{attribute 'enable_dynamic_creation'}
FUNCTION_BLOCK FB_JobEventStream IMPLEMENTS InterfaceJobEventObservable
VAR_INPUT
END_VAR
VAR_OUTPUT
END_VAR
VAR
	_observers : ARRAY[1..ParamFuturesLib.MAX_JOB_EVENT_OBSERVERS] OF InterfaceJobEventObserver;
	_filter_state : E_FutureExecutionState := E_FutureExecutionState.idle;
	_filter_event_type : E_JobEventType := E_JobEventType.TRANSITION;
	_filter_executor_id : T_MaxString := '';
	_filter_error_min : UDINT := 0;
	_filter_error_max : UDINT := 16#FFFFFFFF;
	_filter_enabled : ST_FilterStates;
END_VAR

METHOD ClearFilters : InterfaceJobEventObservable
VAR_INPUT
END_VAR
_filter_enabled.state := FALSE;
_filter_enabled.event_type := FALSE;
_filter_enabled.executor_id := FALSE;
_filter_enabled.error_range := FALSE;
ClearFilters := THIS^;
END_METHOD

METHOD emit_event : BOOL
VAR_INPUT
	event : ST_JobEvent;
END_VAR
VAR
	i : UINT;
	should_emit : BOOL := TRUE;
END_VAR
// フィルター判定
IF _filter_enabled.state AND event.state_new <> _filter_state THEN
	should_emit := FALSE;
END_IF
IF _filter_enabled.event_type AND event.event_type <> _filter_event_type THEN
	should_emit := FALSE;
END_IF
IF _filter_enabled.executor_id AND event.executor_id <> _filter_executor_id THEN
	should_emit := FALSE;
END_IF
IF _filter_enabled.error_range AND (event.error_id < _filter_error_min OR event.error_id > _filter_error_max) THEN
	should_emit := FALSE;
END_IF

// 配信実行
IF should_emit THEN
	FOR i := 1 TO ParamFuturesLib.MAX_JOB_EVENT_OBSERVERS DO
		IF _observers[i] <> 0 THEN
			_observers[i].OnJobEvent(event);
		END_IF
	END_FOR
	emit_event := TRUE;
ELSE
	emit_event := FALSE;
END_IF
END_METHOD

METHOD Subscribe : BOOL
VAR_INPUT
	observer : InterfaceJobEventObserver;
END_VAR
VAR
	i : UINT;
	bSubscribed : BOOL := FALSE;
	idxEmpty : UINT := 0;
END_VAR
IF observer = 0 THEN
	Subscribe := FALSE;
	RETURN;
END_IF

// 既存購読確認と空きスロット検索
FOR i := 1 TO ParamFuturesLib.MAX_JOB_EVENT_OBSERVERS DO
	IF _observers[i] = observer THEN
		bSubscribed := TRUE;
		EXIT;
	END_IF
	IF idxEmpty = 0 AND _observers[i] = 0 THEN
		idxEmpty := i;
	END_IF
END_FOR

IF bSubscribed THEN
	Subscribe := TRUE; // 既に購読済み
ELSIF idxEmpty <> 0 THEN
	_observers[idxEmpty] := observer;
	Subscribe := TRUE;
ELSE
	Subscribe := FALSE; // 配列満杯
END_IF
END_METHOD

METHOD Unsubscribe : BOOL
VAR_INPUT
	observer : InterfaceJobEventObserver;
END_VAR
VAR
	i : UINT;
	bFound : BOOL := FALSE;
END_VAR
IF observer = 0 THEN
	Unsubscribe := FALSE;
	RETURN;
END_IF

FOR i := 1 TO ParamFuturesLib.MAX_JOB_EVENT_OBSERVERS DO
	IF _observers[i] = observer THEN
		_observers[i] := 0; // Observer削除
		bFound := TRUE;
		EXIT;
	END_IF
END_FOR

Unsubscribe := bFound;
END_METHOD

METHOD WhereErrorRange : InterfaceJobEventObservable
VAR_INPUT
	min_error : UDINT;
	max_error : UDINT;
END_VAR
_filter_error_min := min_error;
_filter_error_max := max_error;
_filter_enabled.error_range := TRUE;
WhereErrorRange := THIS^;
END_METHOD

METHOD WhereEventType : InterfaceJobEventObservable
VAR_INPUT
	event_type : E_JobEventType;
END_VAR
_filter_event_type := event_type;
_filter_enabled.event_type := TRUE;
WhereEventType := THIS^;
END_METHOD

METHOD WhereExecutorId : InterfaceJobEventObservable
VAR_INPUT
	executor_id : STRING;
END_VAR
_filter_executor_id := executor_id;
_filter_enabled.executor_id := TRUE;
WhereExecutorId := THIS^;
END_METHOD

METHOD WhereState : InterfaceJobEventObservable
VAR_INPUT
	target_state : E_FutureExecutionState;
END_VAR
_filter_state := target_state;
_filter_enabled.state := TRUE;
WhereState := THIS^;
END_METHOD

END_FUNCTION_BLOCK

(* stored: Version 1.1.0.1, ProductVersion 3.1.4024.15
   POU FB_JobEventStream: Id {b3b0b56f-92ef-4af1-8453-d6abd560995d}, SpecialFunc None
   Method ClearFilters: Id {a7c8f4d3-2e9b-4f8a-b6c5-8d7e6f5a4b3c}
   Method emit_event: Id {f2d1e8a7-3b4c-4529-a6d8-9e7f6d5c4b3a}
   Method Subscribe: Id {3c8f9e4a-5d6b-4728-a19c-8e7f6d5c4b3a}
   Method Unsubscribe: Id {7b9a5e2c-8d4f-4618-b5a7-9c8b7e6d5f4e}
   Method WhereErrorRange: Id {8d7c6b5a-4928-4f17-a6d5-3c2b1a9e8f7d}
   Method WhereEventType: Id {bb7112d7-3363-4ff5-a12e-469d07c34588}
   Method WhereExecutorId: Id {57f7bab4-907d-45ad-b0c3-6453c49a2eca}
   Method WhereState: Id {7989d8ed-b967-4573-8591-9a78b4b7fe98} *)
